(* IEC 61131-3 sources: POMIRTS_lab3/AS/Library_2/AsANSL, 3 files *)

(* ---- AsANSL.typ ---- *)
TYPE
	AsANSLTimeStampType : STRUCT		(*timestamp structure*)
		timeStampSec	: UDINT;		(*seconds since 01.01.1970*)
		timeStampNsec	: UDINT;		(*nanoseconds*)
	END_STRUCT;

	AsANSLClientDiagInfoType : STRUCT					(*client diagnose structure*)
		clientDataObjName	: STRING[256];				(*name of the data object*)
		clientTimeStamp 	: AsANSLTimeStampType;		(*timestamp of last update*)
		clientConn			: UDINT;					(*number of the connections*)
		clientConnErr		: UDINT;					(*number of the connections with error*)
	END_STRUCT;

	AsANSLClientDiagConnInfoType : STRUCT				(*client connection diagnose structure*)
		connName			: STRING[64];				(*name of the connection*)
		connTargetAddr		: STRING[64];				(*address/hostname of the target*)
		connTimeStamp 		: AsANSLTimeStampType;		(*timestamp of last update*)
		connStatus			: UDINT;					(*state of the connection*)
		connError			: UDINT;					(*error of the connection*)
		connPvRead			: UDINT;					(*number of read pv*)
		connPvReadErr		: UDINT;					(*number of read pv with error*)
		connPvWrite			: UDINT;					(*number of write pv*)
		connPvWriteErr		: UDINT;					(*number of write pv with error*)
		connNumReadJobs		: UDINT;					(*read jobs since last initialization*)
		connNumSendJobs		: UDINT;					(*send jobs since last initialization*)
		connNumErr			: UDINT;					(*number of connection error since last initialization*)
	END_STRUCT;

	AsANSLClientDiagRedConnInfoType : STRUCT			(*client redundancy connection diagnose structure*)
		redConnActIpAddr	: STRING[64];				(*ip address of the active used connection*)
		redConnAct 			: UDINT;					(*identify the active used connection*)
		redConnStatus		: UDINT;					(*state of the redundancy connection*)
		redConnCluError		: UDINT;					(*error of the cluster connection*)
		redConnPriError		: UDINT;					(*error of the primary connection*)
		redConnSecError		: UDINT;					(*error of the secondary connection*)
		redConnRRPrio		: UDINT;					(*priority of redundancy relevant connection*)
	END_STRUCT;

	AsANSLClientDiagPvInfoType : STRUCT					(*pv connection diagnose structure*)
		pvNameLocal			: STRING[512];				(*name of the local pv*)
		pvNameRemote		: STRING[512];				(*name of the remote pv*)
		pvTimeStamp 		: AsANSLTimeStampType;		(*timestamp of last update*)
		pvStatus			: UDINT;					(*state of the pv connection*)
		pvError				: UDINT;					(*error of the pv connection*)
		pvDirection			: UDINT;					(*direction of pv - read/write*)
	END_STRUCT;

	AsANSLServerDiagConnInfoType : STRUCT					(*server connection diagnose structure*)
		connClientIpAddr			: STRING[64];			(*ip address of client station*)
		connServerIpAddr			: STRING[64];			(*ip address of used server interface*)
		connTimeStamp				: AsANSLTimeStampType;	(*timestamp when the connetion got established*)
		connTimeout					: UDINT;				(*connection timeout*)
		connSendDelay				: UDINT;				(*connetion send delay*)
		connPort					: UDINT;				(*connection port*)
		connBufferSize				: UDINT;				(*connection buffer size*)
		connServiceObjects			: UDINT;				(*number of registered ANSL service objects*)
		connBytesRecv				: UDINT;				(*number of received bytes*)
		connBytesSent				: UDINT;				(*number of sent bytes*)
		connRequestsRecv			: UDINT;				(*number of received requests*)
		connEventsSent				: UDINT;				(*number of sent events*)
		connResponsesSent			: UDINT;				(*number of sent responses*)
		connEventPvs				: UDINT;				(*number of registered event pvs*)
		connEventPvProcessing 		: BOOL;					(*event processing flag (activated/deactivated)*)
		connEventPvRate				: UDINT;				(*number of event pvs checked per block*)
		connEventPvTime				: UDINT;				(*time to wait between two blocks*)
		connEventPvsChangedBlock	: UDINT;				(*number of pvs changed last block*)
		connEventPvsChangedAll		: UDINT;				(*number of pvs changed overall*)
		connRRPrio					: UDINT;				(*priority of redundancy relevant connection*)
		connRRName					: STRING[64];			(*name of redundancy relevant connection*)
	END_STRUCT;

END_TYPE

(* ---- AsANSL.fun ---- *)
{REDUND_OK} {REDUND_UNREPLICABLE} FUNCTION_BLOCK AsANSLClientStart			(*starts an ANSL client which read and write PVs from other controllers based on the configuration; asynchronous execution*)
	VAR_INPUT
		enable			: BOOL;							(*enables execution*)
		dataObjName		: STRING[256];					(*datamodul name*)
	END_VAR

	VAR_OUTPUT
		status			: UINT;			(*execution status: ERR_OK, ERR_FUB_ENABLE_FALSE, ERR_FUB_BUSY, 0xXXXX = see help*)
	END_VAR

	VAR
        i_state			: UINT;			(*internal variable*)
		i_result		: UINT;			(*internal variable*)
	END_VAR
END_FUNCTION_BLOCK

{REDUND_OK} {REDUND_UNREPLICABLE} FUNCTION_BLOCK AsANSLClientStop		(*stops an ANSL client which read and write PVs from other controllers based on the configuration; asynchronous execution*)
	VAR_INPUT
		enable			: BOOL;							(*enables execution*)
		dataObjName		: STRING[256];					(*datamodul name*)
	END_VAR

	VAR_OUTPUT
		status			: UINT;			(*execution status: ERR_OK, ERR_FUB_ENABLE_FALSE, ERR_FUB_BUSY, 0xXXXX = see help*)
	END_VAR

	VAR
        i_state			: UINT;			(*internal variable*)
		i_result		: UINT;			(*internal variable*)
	END_VAR
END_FUNCTION_BLOCK

{REDUND_OK} {REDUND_UNREPLICABLE} FUNCTION_BLOCK AsANSLClientDiag			(*reads diagnostic infos from an ANSL client; asynchronous execution*)
	VAR_INPUT
		enable			: BOOL;							(*enables execution*)
		dataObjName		: STRING[256];					(*datamodul name*)
	END_VAR

	VAR_OUTPUT
		status			: UINT;							(*execution status: ERR_OK, ERR_FUB_ENABLE_FALSE, ERR_FUB_BUSY, 0xXXXX = see help*)
		ClientDiagInfo	: AsANSLClientDiagInfoType;		(*client info struct*)
	END_VAR

	VAR
        i_state			: UINT;			(*internal variable*)
		i_result		: UINT;			(*internal variable*)
	END_VAR
END_FUNCTION_BLOCK

{REDUND_OK} {REDUND_UNREPLICABLE} FUNCTION_BLOCK AsANSLClientDiagAll		(*reads diagnostic infos from an ANSL client; asynchronous execution*)
	VAR_INPUT
		enable			: BOOL;							(*enables execution*)
		index			: UDINT;						(*index to iterate the clients*)
	END_VAR

	VAR_OUTPUT
		status				: UINT;						(*execution status: ERR_OK, ERR_FUB_ENABLE_FALSE, ERR_FUB_BUSY, 0xXXXX = see help*)
		ClientDiagInfo	: AsANSLClientDiagInfoType;		(*client info struct*)
	END_VAR

	VAR
        i_state			: UINT;			(*internal variable*)
		i_result		: UINT;			(*internal variable*)
	END_VAR
END_FUNCTION_BLOCK

{REDUND_OK} {REDUND_UNREPLICABLE} FUNCTION_BLOCK AsANSLClientDiagConn	(*reads diagnostic infos of a connection of an ANSL client; asynchronous execution*)
	VAR_INPUT
		enable			: BOOL;							(*enables execution*)
		dataObjName		: STRING[256];					(*datamodul name*)
		connName		: STRING[64];					(*connection name*)
	END_VAR

	VAR_OUTPUT
		status				: UINT;								(*execution status: ERR_OK, ERR_FUB_ENABLE_FALSE, ERR_FUB_BUSY, 0xXXXX = see help*)
		ClientDiagConnInfo	: AsANSLClientDiagConnInfoType;		(*client connection info struct*)
	END_VAR

	VAR
        i_state			: UINT;			(*internal variable*)
		i_result		: UINT;			(*internal variable*)
	END_VAR
END_FUNCTION_BLOCK

{REDUND_OK} {REDUND_UNREPLICABLE} FUNCTION_BLOCK AsANSLClientDiagConnAll	(*reads diagnostic infos of a connection of an ANSL client; asynchronous execution*)
	VAR_INPUT
		enable			: BOOL;							(*enables execution*)
		dataObjName		: STRING[256];					(*datamodul name*)
		index			: UDINT;						(*index to iterate the connections*)
		filterOption	: UDINT;						(*options: asANSL_OPTION_FILTER_ALL, asANSL_OPTION_FILTER_NOERROR, asANSL_OPTION_FILTER_ERROR*)
	END_VAR

	VAR_OUTPUT
		status				: UINT;								(*execution status: ERR_OK, ERR_FUB_ENABLE_FALSE, ERR_FUB_BUSY, 0xXXXX = see help*)
		ClientDiagConnInfo	: AsANSLClientDiagConnInfoType;		(*client connection info struct*)
	END_VAR

	VAR
        i_state			: UINT;			(*internal variable*)
		i_result		: UINT;			(*internal variable*)
	END_VAR
END_FUNCTION_BLOCK

{REDUND_OK} {REDUND_UNREPLICABLE} FUNCTION_BLOCK AsANSLClientDiagRedConn	(*reads diagnostic infos of a redundancy connection of an ANSL client; asynchronous execution*)
	VAR_INPUT
		enable			: BOOL;							(*enables execution*)
		dataObjName		: STRING[256];					(*datamodul name*)
		connName		: STRING[64];					(*connection name*)
	END_VAR

	VAR_OUTPUT
		status					: UINT;									(*execution status: ERR_OK, ERR_FUB_ENABLE_FALSE, ERR_FUB_BUSY, 0xXXXX = see help*)
		ClientDiagRedConnInfo	: AsANSLClientDiagRedConnInfoType;		(*client redundancy connection info struct*)
	END_VAR

	VAR
        i_state			: UINT;			(*internal variable*)
		i_result		: UINT;			(*internal variable*)
	END_VAR
END_FUNCTION_BLOCK

{REDUND_OK} {REDUND_UNREPLICABLE} FUNCTION_BLOCK AsANSLClientDiagPv		(*reads diagnostic infos of a pv connection of an ANSL client; asynchronous execution*)
	VAR_INPUT
		enable			: BOOL;							(*enables execution*)
		dataObjName		: STRING[256];					(*datamodul name*)
		connName		: STRING[64];					(*connection name*)
		localPvName		: STRING[512];					(*local pv name given as pointer*)
		remotePvName	: STRING[512];					(*remote pv name given as pointer*)
	END_VAR

	VAR_OUTPUT
		status				: UINT;								(*execution status: ERR_OK, ERR_FUB_ENABLE_FALSE, ERR_FUB_BUSY, 0xXXXX = see help*)
		ClientDiagPvInfo	: AsANSLClientDiagPvInfoType;		(*client pv info struct*)
	END_VAR

	VAR
        i_state			: UINT;			(*internal variable*)
		i_result		: UINT;			(*internal variable*)
	END_VAR
END_FUNCTION_BLOCK

{REDUND_OK} {REDUND_UNREPLICABLE} FUNCTION_BLOCK AsANSLClientDiagPvAll	(*reads diagnostic infos of a pv connection of an ANSL client; asynchronous execution*)
	VAR_INPUT
		enable			: BOOL;							(*enables execution*)
		dataObjName		: STRING[256];					(*datamodul name*)
		connName		: STRING[64];					(*connection name*)
		index			: UDINT;						(*index to iterate the connections*)
		filterOption	: UDINT;						(*options: asANSL_OPTION_FILTER_ALL, asANSL_OPTION_FILTER_NOERROR, asANSL_OPTION_FILTER_ERROR*)
	END_VAR

	VAR_OUTPUT
		status				: UINT;								(*execution status: ERR_OK, ERR_FUB_ENABLE_FALSE, ERR_FUB_BUSY, 0xXXXX = see help*)
		ClientDiagPvInfo	: AsANSLClientDiagPvInfoType;		(*client pv info struct*)
	END_VAR

	VAR
        i_state			: UINT;			(*internal variable*)
		i_result		: UINT;			(*internal variable*)
	END_VAR
END_FUNCTION_BLOCK

{REDUND_OK} {REDUND_UNREPLICABLE} FUNCTION_BLOCK AsANSLServerRRInfo	(*reads infos of the redundancy relevant connections of an ANSL Server; asynchronous execution*)
	VAR_INPUT
		enable					: BOOL;					(*enables execution*)
		pConnList				: UDINT;				(*names of all redundancy relevant connections given as pointer*)
		maxConnListLenght		: UDINT;				(*maximum length of the string (pConnList)*)
		cpuOption				: UDINT;				(*options: asANSL_OPTION_CPU_LOCAL, asANSL_OPTION_CPU_PARTNER*)
	END_VAR

	VAR_OUTPUT
		status						: UINT;				(*execution status: ERR_OK, ERR_FUB_ENABLE_FALSE, ERR_FUB_BUSY, 0xXXXX = see help*)
		connListLenght  			: UDINT;			(*data length of the string (pConnList)*)
		rrConnCount					: UDINT;			(*number of redundancy relevant connections*)
		rrConnIndicator				: UDINT;			(*priority of all redundancy relevant connections*)
	END_VAR

	VAR
        i_state			: UINT;			(*internal variable*)
		i_result		: UINT;			(*internal variable*)
	END_VAR
END_FUNCTION_BLOCK

{REDUND_OK} {REDUND_UNREPLICABLE} FUNCTION AsANSLServerConnCount : UDINT	(*return the number of activ connections of an ANSL Server*)
END_FUNCTION

{REDUND_OK} {REDUND_UNREPLICABLE} FUNCTION_BLOCK AsANSLServerDiagConnAll	(*reads diagnostic infos of an ANSL server connection; asynchronous execution*)
	VAR_INPUT
		enable				: BOOL;						(*enables execution*)
		index				: UDINT;					(*index to iterate the connections*)
		filterClientIpAddr	: STRING[64];				(*filter to list only connections with the same ClientIpAddr*)
	END_VAR

	VAR_OUTPUT
		status				: UINT;								(*execution status: ERR_OK, ERR_FUB_ENABLE_FALSE, ERR_FUB_BUSY, 0xXXXX = see help*)
		ServerDiagConnInfo	: AsANSLServerDiagConnInfoType;		(*server connection info struct*)
	END_VAR

	VAR
        i_state			: UINT;			(*internal variable*)
		i_result		: UINT;			(*internal variable*)
	END_VAR
END_FUNCTION_BLOCK

(* ---- AsANSL.var ---- *)
VAR CONSTANT
	asANSL_OPTION_FILTER_ALL 			: USINT		:= 0;		(*iterate over all connections*)
	asANSL_OPTION_FILTER_NOERROR 		: USINT		:= 1;		(*iterate over all connections without error*)
	asANSL_OPTION_FILTER_ERROR			: USINT		:= 2;		(*iterate over all connections with error*)

	asANSL_OPTION_CPU_LOCAL				: USINT		:= 0;		(*local plc*)
	asANSL_OPTION_CPU_PARTNER			: USINT		:= 1;		(*partner plc*)

	asANSL_PV_DIRECTION_READ			: USINT		:= 1;		(*client read pv*)
	asANSL_PV_DIRECTION_WRITE			: USINT		:= 2;		(*client write pv*)

	asANSL_RED_CONN_NO_CONNECTION		: UDINT		:= 0;		(*no connection to one of the redundancy CPUs*)
	asANSL_RED_CONN_PRI_NOT_ACTIV		: UDINT		:= 2;		(*connection of the primary (not activ) CPU*)
	asANSL_RED_CONN_PRI_ACTIV			: UDINT		:= 3;		(*connection of the primary (activ) CPU*)
	asANSL_RED_CONN_SEC_NOT_ACTIV 		: UDINT		:= 4;		(*connection of the secondary (not activ) CPU*)
	asANSL_RED_CONN_SEC_ACTIV			: UDINT		:= 5;		(*connection of the secondary (activ) CPU*)

	asANSL_RED_CONN_CLU_OK				: UDINT		:= 1;		(*cluster connection is OK*)
	asANSL_RED_CONN_CLU_ERROR			: UDINT		:= 2;		(*cluster connection is in an error state*)
	asANSL_RED_CONN_PRI_OK				: UDINT		:= 4;		(*connection to the primary CPU is OK*)
	asANSL_RED_CONN_PRI_ERROR			: UDINT		:= 8;		(*connection to the primary CPU is in an error state*)
	asANSL_RED_CONN_SEC_OK				: UDINT		:= 16;		(*connection to the secondary CPU is OK*)
	asANSL_RED_CONN_SEC_ERROR			: UDINT		:= 32;		(*connection to the secondary CPU is in an error state*)

	asANSL_ERR_MEMORY_RESOURCE			: UINT		:= 31651;	(*system out of memory*)
	asANSL_ERR_EVENT_RESOURCE			: UINT		:= 31652;	(*system out of event resource*)
	asANSL_ERR_THREAD_RESOURCE			: UINT		:= 31653;	(*system out of thread resource*)
	asANSL_ERR_SYNC_RESOURCE			: UINT		:= 31654;	(*system out of synchronisation resource*)
	asANSL_ERR_FILE_RESOURCE			: UINT		:= 31655;	(*system out of file resource*)

	asANSL_ERR_PARAM_INVALID			: UINT		:= 31870;	(*invalid parameter*)
	asANSL_ERR_XML_PARSER_INIT_ERROR	: UINT		:= 31871;	(*xml parser error*)
	asANSL_ERR_XML_INVALID				: UINT		:= 31872;	(*invalid xml configuration*)
	asANSL_ERR_DATAMODUL_NOT_EXIST		: UINT		:= 31873;	(*datamodul not found*)
	asANSL_ERR_CLIENT_NOT_EXIST			: UINT		:= 31874;	(*client not found/started*)
	asANSL_ERR_CONN_NOT_EXIST			: UINT		:= 31875;	(*connection not found*)
	asANSL_ERR_PV_CONN_NOT_EXIST		: UINT		:= 31876;	(*pv connection not found*)
	asANSL_ERR_END_OF_LIST				: UINT		:= 31877;	(*end of client/connection/pv list*)
END_VAR
